(****************************************************************************************************)
(*							Beckhoff Automation Poland												*)
(*							FB_ReceipRW v1.1														*)
(*									17.09.2012														*)
(*		Blok funkcyjny zapisu i odczytu receptury (dowolnej zmiennej) w formie binarnej				*)
(*____________________________________________________________________________________________________
	Versions:
		v1.1	05.08.2016	* Przepisana wersja do TwinCat3
		v1.0	17.09.2012	* Podstawowa wersja z TwinCat2
____________________________________________________________________________________________________*)
FUNCTION_BLOCK FB_ReceipRW
VAR_INPUT
	sNetId			: T_AmsNetId;
	sPath			: STRING;
	sFileName		: STRING;
	bSave			: BOOL;
	pWriteBuff		: DWORD;
	cbWriteLen		: UDINT;
	bLoad			: BOOL;
	pReadBuff		: DWORD;
	cbReadLen		: UDINT;
END_VAR
VAR_OUTPUT
	bBusy			: BOOL;
	bError			: BOOL;
END_VAR
VAR
	rtSave			: R_TRIG;
	rtLoad			: R_TRIG;
	bSaveAction		: BOOL;
	bLoadAction		: BOOL;
	fbFileOpen		: FB_FileOpen;
	ftOpen			: F_TRIG;
	fbFileWrite		: FB_FileWrite;
	ftWrite			: F_TRIG;
	fbFileRead		: FB_FileRead;
	ftRead			: F_TRIG;
	fbFileClose		: FB_FileClose;
	ftClose			: F_TRIG;
	rtError			: R_TRIG;
END_VAR

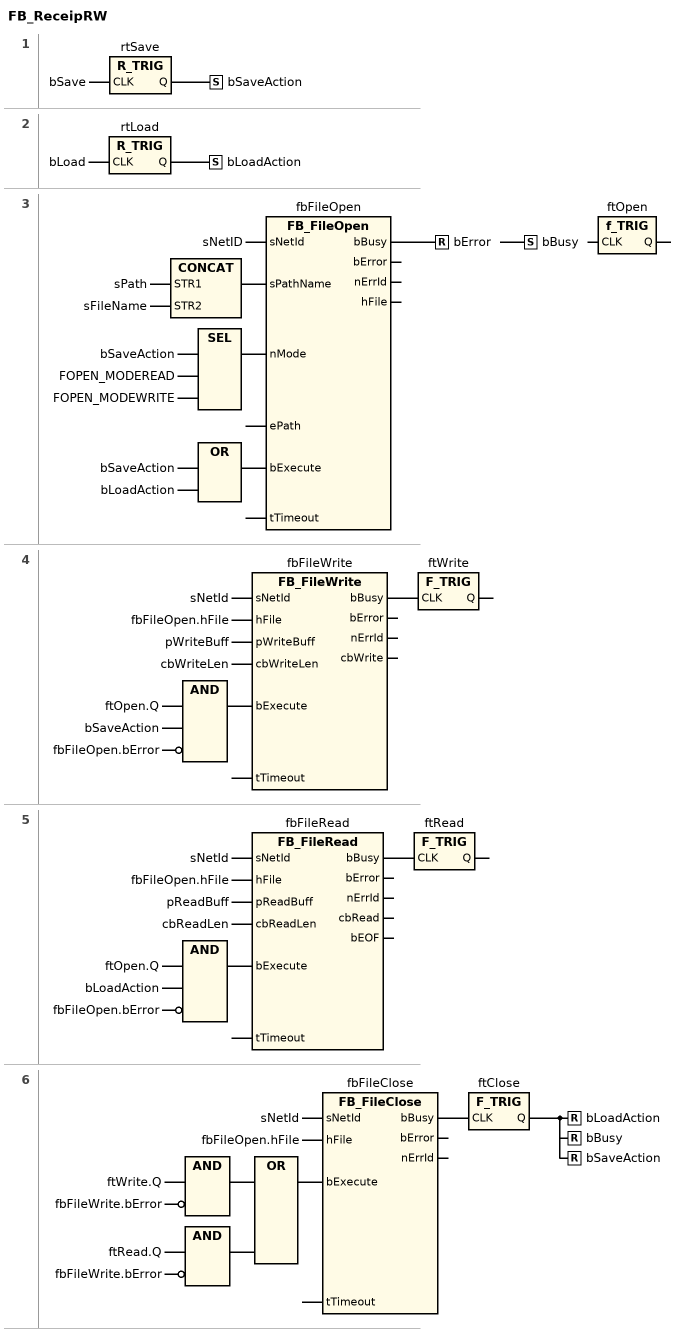
// NETWORK 1
rtSave(CLK := bSave); // R_TRIG
bSaveAction S= rtSave.Q;

// NETWORK 2
rtLoad(CLK := bLoad); // R_TRIG
bLoadAction S= rtLoad.Q;

// NETWORK 3
fbFileOpen(
    sNetId := sNetID,
    sPathName := CONCAT(STR1 := sPath, STR2 := sFileName),
    nMode := SEL(bSaveAction, FOPEN_MODEREAD, FOPEN_MODEWRITE),
    bExecute := bSaveAction OR bLoadAction); // FB_FileOpen
bError R= fbFileOpen.bBusy;
bBusy S= fbFileOpen.bBusy;
ftOpen(CLK := fbFileOpen.bBusy); // f_TRIG

// NETWORK 4
fbFileWrite(
    sNetId := sNetId,
    hFile := fbFileOpen.hFile,
    pWriteBuff := pWriteBuff,
    cbWriteLen := cbWriteLen,
    bExecute := ftOpen.Q AND bSaveAction AND NOT fbFileOpen.bError); // FB_FileWrite
ftWrite(CLK := fbFileWrite.bBusy); // F_TRIG

// NETWORK 5
fbFileRead(
    sNetId := sNetId,
    hFile := fbFileOpen.hFile,
    pReadBuff := pReadBuff,
    cbReadLen := cbReadLen,
    bExecute := ftOpen.Q AND bLoadAction AND NOT fbFileOpen.bError); // FB_FileRead
ftRead(CLK := fbFileRead.bBusy); // F_TRIG

// NETWORK 6
fbFileClose(
    sNetId := sNetId,
    hFile := fbFileOpen.hFile,
    bExecute := ftWrite.Q AND NOT fbFileWrite.bError OR ftRead.Q AND NOT fbFileWrite.bError); // FB_FileClose
ftClose(CLK := fbFileClose.bBusy); // F_TRIG
bLoadAction R= ftClose.Q;
bBusy R= ftClose.Q;
bSaveAction R= ftClose.Q;

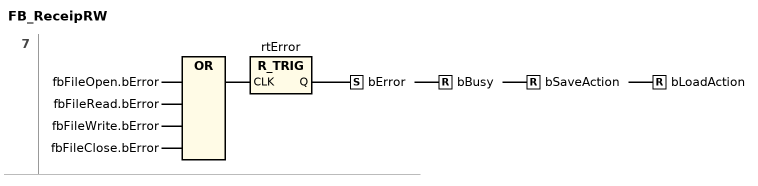
// NETWORK 7
rtError(CLK := fbFileOpen.bError OR fbFileRead.bError OR fbFileWrite.bError OR fbFileClose.bError); // R_TRIG
bError S= rtError.Q;
bBusy R= rtError.Q;
bSaveAction R= rtError.Q;
bLoadAction R= rtError.Q;

END_FUNCTION_BLOCK

(* stored: Version 1.1.0.1, ProductVersion 3.1.4020.3
   POU FB_ReceipRW: Id {4c0cc621-833e-490b-8594-526f54d599df}, SpecialFunc None *)
